FUNCTION_BLOCK FB_Integrator
VAR_INPUT
	ssMethodType: SINT;
	fSignal: LREAL;
END_VAR
VAR_OUTPUT
	fSignalIntegrated: LREAL;
END_VAR
VAR
	c_DiscreteTimeIntegrator_DS: LREAL;
END_VAR



CASE ssMethodType OF
    SS_INITIALIZE: 
        (* SystemInitialize for Atomic SubSystem: '<Root>/Integrator' *)
        (* InitializeConditions for DiscreteIntegrator: '<S1>/Discrete-Time Integrator' *)
        c_DiscreteTimeIntegrator_DS := 0.0;
        (* End of SystemInitialize for SubSystem: '<Root>/Integrator' *)
    SS_STEP: 
        (* Outputs for Atomic SubSystem: '<Root>/Integrator' *)
        (* Outport: '<Root>/fSignalIntegrated' incorporates:
         *  DiscreteIntegrator: '<S1>/Discrete-Time Integrator' *)
        fSignalIntegrated := c_DiscreteTimeIntegrator_DS;
        (* Update for DiscreteIntegrator: '<S1>/Discrete-Time Integrator' *)
        c_DiscreteTimeIntegrator_DS := (0.001 * fSignal) + c_DiscreteTimeIntegrator_DS;
        (* End of Outputs for SubSystem: '<Root>/Integrator' *)
END_CASE;

END_FUNCTION_BLOCK

(* stored: Version 1.1.0.1, ProductVersion 3.1.4024.12
   POU FB_Integrator: Id {ba388259-306e-40da-af33-c63428464cb8}, SpecialFunc None *)
